(* PLC project Unnamed, Unknown Unnamed 1 *)
(* stored: creationDateTime 2026-05-05T00:50:54, modificationDateTime 2026-05-05T00:50:54 *)

(* simple boolean *)
PROGRAM main
  VAR
    SwitchA : BOOL := TRUE;
    SwitchB : BOOL := FALSE;
    Light : BOOL := FALSE;
  END_VAR

            Light := SwitchA AND SwitchB;
          
END_PROGRAM

PROGRAM temp_sensor
  VAR_INPUT
    TempSensor1 : DINT;
    TempSensor2 : DINT;
  END_VAR
  VAR_OUTPUT
    Fan : BOOL;
  END_VAR

            Fan := TempSensor1 > TempSensor2;
          
END_PROGRAM

CONFIGURATION Config0
  RESOURCE Res0 ON PLC
    TASK task0(INTERVAL := T#20ms, PRIORITY := 1);
    TASK task1(INTERVAL := T#20ms, PRIORITY := 1);
    PROGRAM instance0 WITH task0 : main;
    PROGRAM instance1 WITH task1 : temp_sensor;
  END_RESOURCE
END_CONFIGURATION
